Universal Robots PolyScope program: box_search.urp

Program box_search (installation=default directory=/programs createdIn=5.10.0.106288 lastSavedIn=5.10.0.106288 robotSerialNumber=20185500256)
Calibrated DH parameters: a=[0.000163, -0.146131, -0.38577, 0.000126, -0.000021, 0]; d=[0.161954, 188.306531, -157.478086, -30.695088, 0.099716, 0.099628]; alpha=[1.569701, -0.00212, 0.002263, 1.570438, -1.570123, 0]; deltaTheta=[0, -1.219859, 7.681919, -0.178877, -0.000001, 0]
Robot Program (runOnlyOnce=true)
  box := [[0,0],[0,0]]
  MoveL speed 250 mm/s, acceleration 1200 mm/s^2 (useActiveTCP=true) feature=Base
    Waypoint starting_point: TCP in base x=182.547 y=-305.825 z=46.754 mm, rx=-0.0132 ry=3.0946 rz=0.0237 rad; joints [95.869, -107.252, 132.922, -115.024, -87.078, 5.465] deg; TCP offset x=0 y=0 z=250.5 mm, rx=0 ry=0 rz=0 rad
  Loop Counting (count=2) loopVariable(name=Loop_1)
    axis := Loop_1
    Loop Counting (count=2) loopVariable(name=Loop_2)
      direction := Loop_2 % 2
      If direction
        delta := 1
      Else 
        delta := -1
      box_border := p_rel_1D(get_actual_tcp_pose(), delta, axis)
      MoveL speed 50 mm/s, acceleration 300 mm/s^2 (useActiveTCP=true) feature=Base
        Waypoint Waypoint (Variable): variable=box_border
          Until TOOL_CONTACT_DETECTION (allowActions=true retraction=0.001 decelerationAcceleration=1.5 decelerationAngularAcceleration=34.906585)
            coordinate := get_actual_tcp_pose()
            Script: box[axis, direction] = coordinate[axis]
  URCap XML-RPC Call (DTI UR Helper, Danish Technological Institute) dataModel(xmlrpc_function=set_box_coordinates, xmlrpc_handle=calibration); state(isChildrenLocked=true)
    succes := calibration.set_box_coordinates(box[0,0], box[0,1], box[1,0], box[1,1])
